(* PLC project Unnamed, Unknown Unnamed 1 *)
(* stored: creationDateTime 2024-03-02T19:19:35, modificationDateTime 2024-03-02T20:00:20 *)

PROGRAM CybICS
  VAR
    systemSen AT %IX0.1 : BOOL := 0;
    boSen AT %IX0.2 : BOOL := 0;
    heartbeat AT %QX0.0 : BOOL := 0;
    compressor AT %QX0.1 : BOOL := 0;
    systemValve AT %QX0.2 : BOOL := 0;
    gstSig AT %QX0.3 : BOOL := 0;
    gst AT %MW100 : UINT;
    hpt AT %MW102 : UINT := 0;
    stop AT %MW104 : UINT := 0;
    manual AT %MW106 : UINT := 0;
    compressorState AT %MW200 : UINT := 0;
    countHeartbeat AT %MW400 : UINT := 0;
  END_VAR

              (* System heartbeat *)
  IF countHeartbeat < 20 THEN 
    heartbeat := FALSE;    
  ELSIF countHeartbeat < 40 THEN
    heartbeat := TRUE;
  ELSE
    countHeartbeat := 0;
  END_IF;
  
  (* System running state *)
  IF stop < 1 THEN
    (* System running in automatic mode *)
    IF manual < 1 THEN
      (* Refill GST, when below 60 and fill it up to 254 *)
      IF gst < 60 AND countHeartbeat = 0 THEN
        countHeartbeat := 1;
      ELSIF gst < 240 AND countHeartbeat = 1 THEN
        countHeartbeat := 1;
      ELSE
        countHeartbeat := 0;
      END_IF;      

      (* Run compressor when below 60 and fill it up to 89 *)
      (* Only run compressor, when GST > 50 *)
      IF hpt < 60 AND compressorState = 0 AND gst > 50 THEN    
        compressorState := 1;
      ELSIF hpt < 90 AND compressorState = 1 AND gst > 50 THEN    
        compressorState := 1;
      ELSE
        compressorState := 0;
      END_IF;
  
  
      IF hpt > 50 AND hpt<100 THEN
        systemValve := TRUE;
      ELSE
        systemValve := FALSE;
      END_IF;
  
      IF compressorState = 1 THEN
        compressor := TRUE;
      ELSE
        compressor := FALSE;
      END_IF;

      IF countHeartbeat = 1 THEN
        gstSig := TRUE;
      ELSE
        gstSig := FALSE;
      END_IF;
      (* ELSE System running in manual mode *)  
    END_IF;
  (* System stop state *)
  ELSE
    compressorState := 0;
    compressor := FALSE;
    systemValve := FALSE;
    countHeartbeat := 0;
    gstSig := FALSE;
  END_IF;
  
  (* Increase the counters *)
  countHeartbeat := countHeartbeat + 1;



          
END_PROGRAM

CONFIGURATION Config0
  RESOURCE Res0 ON PLC
    TASK task0(INTERVAL := T#20ms, PRIORITY := 0);
    PROGRAM instance0 WITH task0 : CybICS;
  END_RESOURCE
END_CONFIGURATION
